# EPICS autosave request: autosave/galil_analog_out.req
$(P)$(R)Deadb_SP
$(P)$(R)_SP
